// SIMATIC STEP 7 (V5.x) project PLC_DVG
// CPU: CPU 317-2 PN/DP
// station: Hardware
// station: SIMATIC 300 Station
// station: P_ADR_BUS
// station: _S7H_BUSSYSTEM_CT
// program: S7 Program(2)

SYMBOL_TABLE
"netsend"	DB 1000	DB 1000
"DI_DO_STATE"	FB 1	FB 1
"TCON"	FB 65	FB 65	// Connect
"TCP_MB_CLIENT"	FB 70	FB 70
"TCP_MB_SERVER"	FB 71	FB 71
"DO_MANUAL"	FC 1	FC 1
"sp_nm11"	I 0.0	BOOL
"md_znm12"	I 0.1	BOOL
"md_nm11"	I 0.2	BOOL
"tz_znm12"	I 0.3	BOOL
"tz_nm11"	I 0.4	BOOL
"sp_nm13"	I 0.5	BOOL
"sp_znm12"	I 0.6	BOOL
"md_nm13"	I 0.7	BOOL
"tz_nm13"	I 1.0	BOOL
"alm_znm15"	I 1.1	BOOL
"sp_nm14"	I 1.2	BOOL
"md_znm15"	I 1.3	BOOL
"md_nm14"	I 1.4	BOOL
"tz_nm14"	I 1.6	BOOL
"md_nm16"	I 2.0	BOOL
"tz_nm17_1"	I 2.1	BOOL
"tz_nm16"	I 2.2	BOOL
"sp_nm17_1"	I 2.4	BOOL
"md_nm17_2"	I 2.5	BOOL
"md_nm17_1"	I 2.6	BOOL
"tz_nm17_2"	I 2.7	BOOL
"sp_nm18"	I 3.0	BOOL
"md_nm19"	I 3.1	BOOL
"md_nm18"	I 3.2	BOOL
"tz_nm19"	I 3.3	BOOL
"tz_nm18"	I 3.4	BOOL
"md_nm19_1"	I 3.7	BOOL
"tz_nm19_1"	I 4.0	BOOL
"sp_no21"	I 4.1	BOOL
"sp_nm20"	I 4.2	BOOL
"md_no21"	I 4.3	BOOL
"md_nm20"	I 4.4	BOOL
"tz_no21"	I 4.5	BOOL
"tz_nm20"	I 4.6	BOOL
"md_no22"	I 5.0	BOOL
"av_vn2"	I 5.1	BOOL
"tz_no22"	I 5.2	BOOL
"md_vn1"	I 5.3	BOOL
"md_vn2"	I 5.4	BOOL
"tz_vn1"	I 5.5	BOOL
"tz_vn2"	I 5.6	BOOL
"sp_vn1"	I 5.7	BOOL
"av_vn1"	I 6.0	BOOL
"md_nv23"	I 6.1	BOOL
"tz_nv23"	I 6.3	BOOL
"temp_vn1"	I 6.4	BOOL
"sp_nv23_1"	I 6.5	BOOL
"sp_nv23"	I 6.6	BOOL
"md_nv23_1"	I 6.7	BOOL
"tz_nv23_1"	I 7.0	BOOL
"sp_nv25"	I 7.1	BOOL
"sp_nm24"	I 7.2	BOOL
"md_nv25"	I 7.3	BOOL
"md_nm24"	I 7.4	BOOL
"tz_nv25"	I 7.5	BOOL
"tz_nm24"	I 7.6	BOOL
"sp_nv26"	I 7.7	BOOL
"md_nv26"	I 8.0	BOOL
"tz_nv27"	I 8.1	BOOL
"tz_nv26"	I 8.2	BOOL
"sp_nv28"	I 8.3	BOOL
"sp_nv27"	I 8.4	BOOL
"md_nv28"	I 8.5	BOOL
"md_nv27"	I 8.6	BOOL
"tz_nv28"	I 8.7	BOOL
"md_nm30"	I 9.1	BOOL
"md_nv29"	I 9.2	BOOL
"tz_nm30"	I 9.3	BOOL
"tz_nv29"	I 9.4	BOOL
"sp_nm31"	I 9.5	BOOL
"md_nm31"	I 9.7	BOOL
"tz_nm31"	I 10.0	BOOL
"md_nc33"	I 10.3	BOOL
"md_nc32"	I 10.4	BOOL
"tz_nc33"	I 10.5	BOOL
"tz_nc32"	I 10.6	BOOL
"sp_nc34"	I 10.7	BOOL
"md_nc34"	I 11.0	BOOL
"tz_nc35"	I 11.1	BOOL
"tz_nc34"	I 11.2	BOOL
"sp_nc35"	I 11.4	BOOL
"md_nc33_1"	I 11.5	BOOL
"md_nc35"	I 11.6	BOOL
"tz_nc33_1"	I 11.7	BOOL
"md_vn3"	I 12.0	BOOL
"tz_vn3"	I 12.2	BOOL
"temp_vn3"	I 12.3	BOOL
"sp_vn3"	I 12.4	BOOL
"av_vn3"	I 12.6	BOOL
"md_dm2"	I 12.7	BOOL
"tz_dm2"	I 13.0	BOOL
"sp_m5"	I 13.1	BOOL
"sp_m4"	I 13.2	BOOL
"md_m5"	I 13.3	BOOL
"md_m4"	I 13.4	BOOL
"tz_m5"	I 13.5	BOOL
"tz_m4"	I 13.6	BOOL
"sp_m6"	I 13.7	BOOL
"md_m6"	I 14.0	BOOL
"tz_m6"	I 14.2	BOOL
"sp_m7"	I 14.4	BOOL
"md_m8"	I 14.5	BOOL
"md_m7"	I 14.6	BOOL
"tz_m8"	I 14.7	BOOL
"sp_c8"	I 15.0	BOOL
"md_c9"	I 15.1	BOOL
"md_c8"	I 15.2	BOOL
"tz_c9"	I 15.3	BOOL
"tz_c8"	I 15.4	BOOL
"sp_c9"	I 15.6	BOOL
"md_ds3"	I 15.7	BOOL
"sp_ds3"	I 16.0	BOOL
"sp_em3"	I 16.1	BOOL
"md_em3"	I 16.3	BOOL
"md_ft1"	I 16.4	BOOL
"tz_em3"	I 16.5	BOOL
"tz_ft1"	I 16.6	BOOL
"md_d2"	I 17.0	BOOL
"tz_vv6"	I 17.1	BOOL
"tz_d2"	I 17.2	BOOL
"sp_zm2"	I 17.3	BOOL
"sp_vv6"	I 17.4	BOOL
"md_zm2"	I 17.5	BOOL
"md_vv6"	I 17.6	BOOL
"tz_zm2"	I 17.7	BOOL
"sp_vd1"	I 18.0	BOOL
"tz_vn5"	I 18.1	BOOL
"md_vd1"	I 18.2	BOOL
"sp_vn5"	I 18.3	BOOL
"tz_vd1"	I 18.4	BOOL
"av_vn5"	I 18.5	BOOL
"md_vn5"	I 18.6	BOOL
"temp_vn5"	I 19.0	BOOL
"sp_vd3"	I 19.1	BOOL
"sp_vd2"	I 19.2	BOOL
"md_vd3"	I 19.3	BOOL
"md_vd2"	I 19.4	BOOL
"tz_vd3"	I 19.5	BOOL
"tz_vd2"	I 19.6	BOOL
"sp_vd4"	I 19.7	BOOL
"md_vd4"	I 20.0	BOOL
"tz_vd5"	I 20.1	BOOL
"tz_vd4"	I 20.2	BOOL
"sp_vd6"	I 20.3	BOOL
"md_vd6"	I 20.5	BOOL
"md_vd5"	I 20.6	BOOL
"tz_vd6"	I 20.7	BOOL
"md_vn4"	I 24.5	BOOL
"tz_vn4"	I 24.7	BOOL
"sp_vn4"	I 25.0	BOOL
"av_vn4"	I 25.2	BOOL
"ZNM15_manual"	M 2000.1	BOOL
"ZNM12_manual"	M 2000.2	BOOL
"ZNM12_pusk_nya"	M 4116.0	BOOL
"ZNM12_stop_nya"	M 4116.1	BOOL
"ZNM15_pusk_nya"	M 4116.2	BOOL
"ZNM15_stop_nya"	M 4116.3	BOOL
"tstArray[0]"	MB 5000	BYTE
"tstArray[1]"	MB 5001	BYTE
"tstArray[2]"	MB 5002	BYTE
"tstArray[3]"	MB 5003	BYTE
"QNM11"	Q 0.0	BOOL
"QZNM15"	Q 0.1	BOOL
"QZNM12"	Q 0.2	BOOL
"QNM16"	Q 0.3	BOOL
"QNM13"	Q 0.4	BOOL
"QNM17_1"	Q 0.5	BOOL
"QNM14"	Q 0.6	BOOL
"QNM17_2"	Q 0.7	BOOL
"QNM18"	Q 1.0	BOOL
"QNO21"	Q 1.1	BOOL
"QNM19"	Q 1.2	BOOL
"QNO22"	Q 1.3	BOOL
"QNM19_1"	Q 1.4	BOOL
"QVN2"	Q 1.5	BOOL
"QNM20"	Q 1.6	BOOL
"QVN1"	Q 1.7	BOOL
"QNV23"	Q 2.0	BOOL
"QNV26"	Q 2.1	BOOL
"QNV23_1"	Q 2.2	BOOL
"QNV27"	Q 2.3	BOOL
"QNM24"	Q 2.4	BOOL
"QNV28"	Q 2.5	BOOL
"QNV25"	Q 2.6	BOOL
"QNV29"	Q 2.7	BOOL
"QNM30"	Q 3.0	BOOL
"QNC34"	Q 3.1	BOOL
"QNM31"	Q 3.2	BOOL
"QNC35"	Q 3.3	BOOL
"QNC32"	Q 3.4	BOOL
"QNC33_1"	Q 3.5	BOOL
"QNC33"	Q 3.6	BOOL
"QVN3"	Q 3.7	BOOL
"QDM2"	Q 4.0	BOOL
"QM7"	Q 4.1	BOOL
"QM4"	Q 4.2	BOOL
"QM8"	Q 4.3	BOOL
"QM5"	Q 4.4	BOOL
"QC8"	Q 4.5	BOOL
"QM6"	Q 4.6	BOOL
"QC9"	Q 4.7	BOOL
"QDS3"	Q 5.0	BOOL
"QVV6"	Q 5.1	BOOL
"QFT1"	Q 5.2	BOOL
"QZM2"	Q 5.3	BOOL
"QEM3"	Q 5.4	BOOL
"QVD1"	Q 5.5	BOOL
"QD2"	Q 5.6	BOOL
"QVN5"	Q 5.7	BOOL
"QVD2"	Q 6.0	BOOL
"QVD6"	Q 6.1	BOOL
"QVD3"	Q 6.2	BOOL
"QVD4"	Q 6.4	BOOL
"QVD5"	Q 6.6	BOOL
"QVN4"	Q 7.7	BOOL
"TON"	SFB 4	SFB 4	// Generate an On Delay
"GET"	SFB 14	SFB 14	// Read Data From a Remote CPU
"PUT"	SFB 15	SFB 15	// Write Data to a Remote CPU
"VAT_DVG_ALL"	VAT 1	
"VAT_2"	VAT 2	
"VAT_3"	VAT 3	
END_SYMBOL_TABLE

FUNCTION_BLOCK "DI_DO_STATE"	// FB 1
TITLE = DI_DO_STATE
//Состояние дискретных входов PLC_DVG для SCADA
VERSION : 0.1
BEGIN
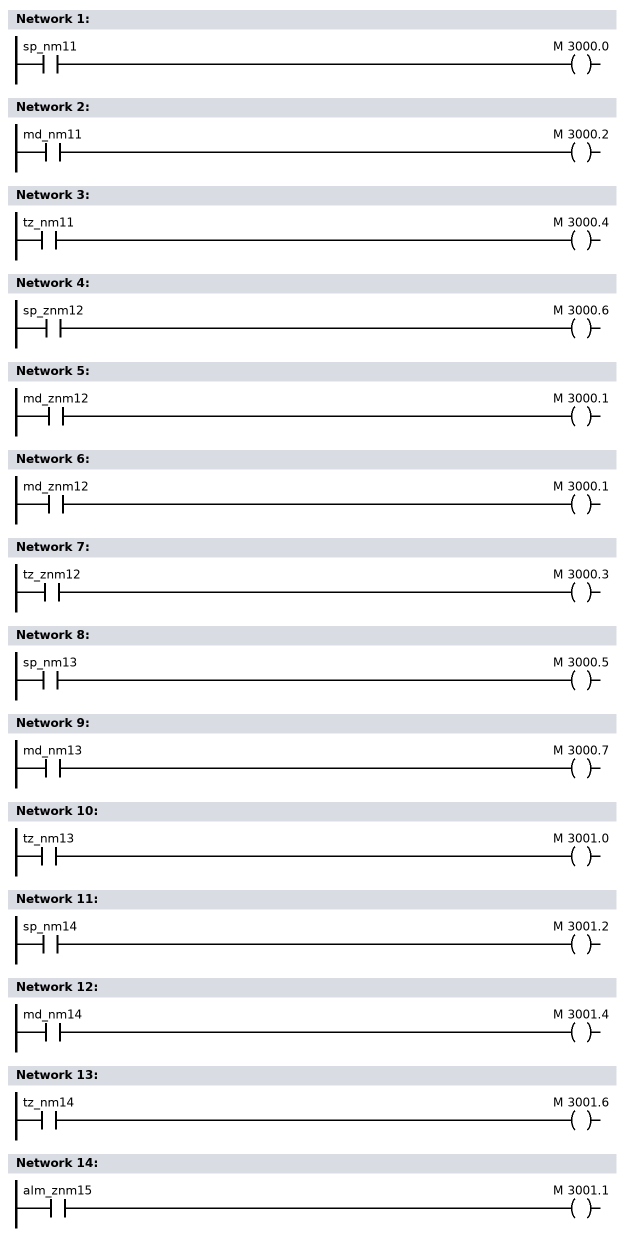
NETWORK
TITLE =
      A     "sp_nm11";
      =     M 3000.0;
NETWORK
TITLE =
      A     "md_nm11";
      =     M 3000.2;
NETWORK
TITLE =
      A     "tz_nm11";
      =     M 3000.4;
NETWORK
TITLE =
      A     "sp_znm12";
      =     M 3000.6;
NETWORK
TITLE =
      A     "md_znm12";
      =     M 3000.1;
NETWORK
TITLE =
      A     "md_znm12";
      =     M 3000.1;
NETWORK
TITLE =
      A     "tz_znm12";
      =     M 3000.3;
NETWORK
TITLE =
      A     "sp_nm13";
      =     M 3000.5;
NETWORK
TITLE =
      A     "md_nm13";
      =     M 3000.7;
NETWORK
TITLE =
      A     "tz_nm13";
      =     M 3001.0;
NETWORK
TITLE =
      A     "sp_nm14";
      =     M 3001.2;
NETWORK
TITLE =
      A     "md_nm14";
      =     M 3001.4;
NETWORK
TITLE =
      A     "tz_nm14";
      =     M 3001.6;
NETWORK
TITLE =
      A     "alm_znm15";
      =     M 3001.1;
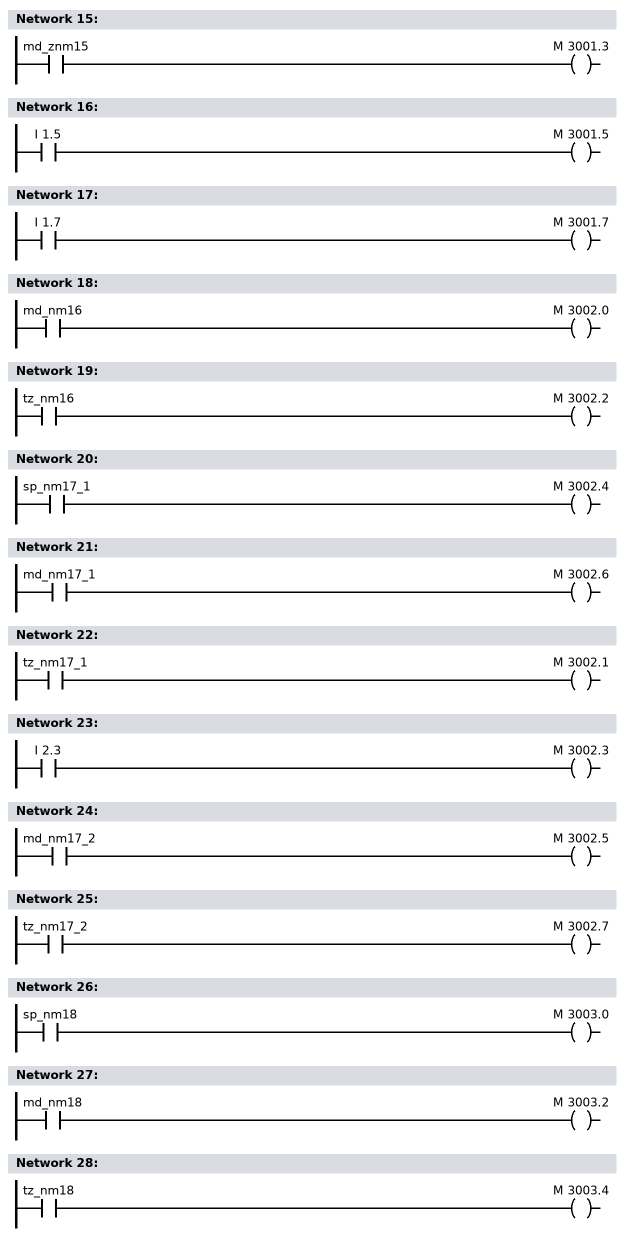
NETWORK
TITLE =
      A     "md_znm15";
      =     M 3001.3;
NETWORK
TITLE =
      A     I 1.5;
      =     M 3001.5;
NETWORK
TITLE =
      A     I 1.7;
      =     M 3001.7;
NETWORK
TITLE =
      A     "md_nm16";
      =     M 3002.0;
NETWORK
TITLE =
      A     "tz_nm16";
      =     M 3002.2;
NETWORK
TITLE =
      A     "sp_nm17_1";
      =     M 3002.4;
NETWORK
TITLE =
      A     "md_nm17_1";
      =     M 3002.6;
NETWORK
TITLE =
      A     "tz_nm17_1";
      =     M 3002.1;
NETWORK
TITLE =
      A     I 2.3;
      =     M 3002.3;
NETWORK
TITLE =
      A     "md_nm17_2";
      =     M 3002.5;
NETWORK
TITLE =
      A     "tz_nm17_2";
      =     M 3002.7;
NETWORK
TITLE =
      A     "sp_nm18";
      =     M 3003.0;
NETWORK
TITLE =
      A     "md_nm18";
      =     M 3003.2;
NETWORK
TITLE =
      A     "tz_nm18";
      =     M 3003.4;
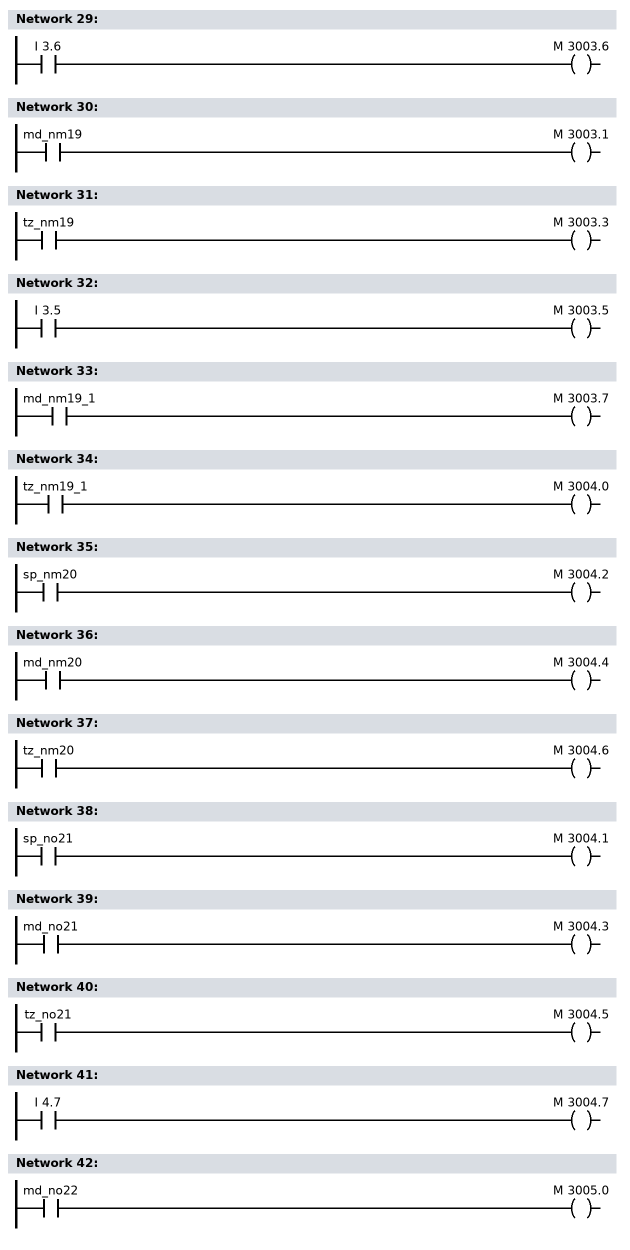
NETWORK
TITLE =
      A     I 3.6;
      =     M 3003.6;
NETWORK
TITLE =
      A     "md_nm19";
      =     M 3003.1;
NETWORK
TITLE =
      A     "tz_nm19";
      =     M 3003.3;
NETWORK
TITLE =
      A     I 3.5;
      =     M 3003.5;
NETWORK
TITLE =
      A     "md_nm19_1";
      =     M 3003.7;
NETWORK
TITLE =
      A     "tz_nm19_1";
      =     M 3004.0;
NETWORK
TITLE =
      A     "sp_nm20";
      =     M 3004.2;
NETWORK
TITLE =
      A     "md_nm20";
      =     M 3004.4;
NETWORK
TITLE =
      A     "tz_nm20";
      =     M 3004.6;
NETWORK
TITLE =
      A     "sp_no21";
      =     M 3004.1;
NETWORK
TITLE =
      A     "md_no21";
      =     M 3004.3;
NETWORK
TITLE =
      A     "tz_no21";
      =     M 3004.5;
NETWORK
TITLE =
      A     I 4.7;
      =     M 3004.7;
NETWORK
TITLE =
      A     "md_no22";
      =     M 3005.0;
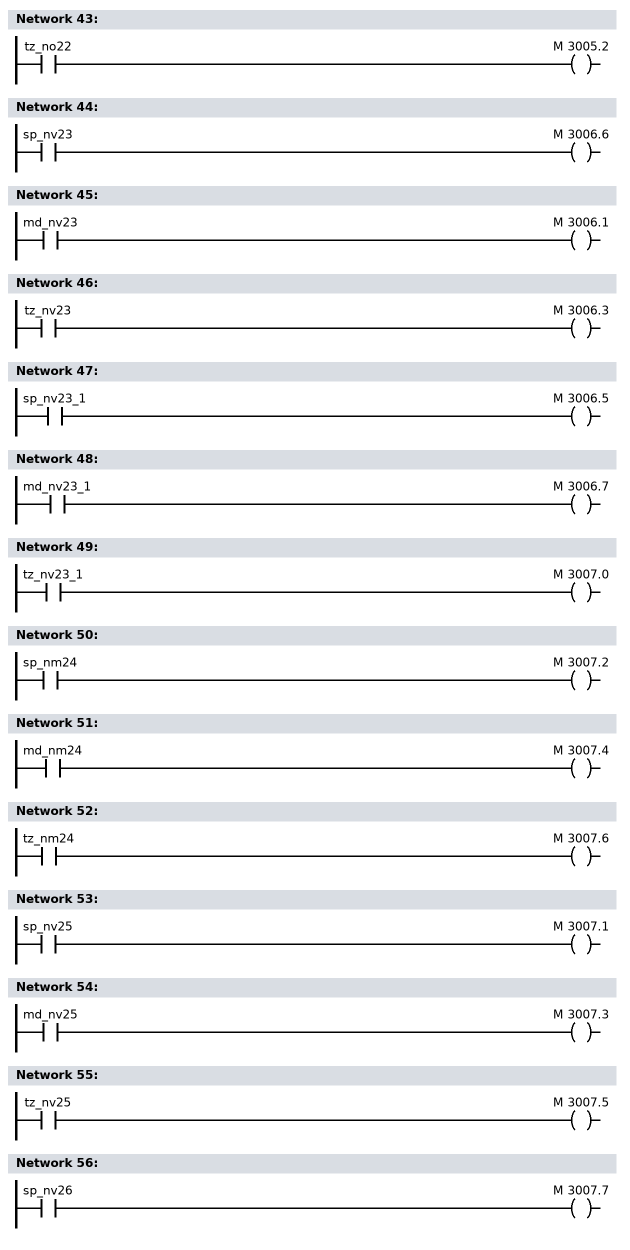
NETWORK
TITLE =
      A     "tz_no22";
      =     M 3005.2;
NETWORK
TITLE =
      A     "sp_nv23";
      =     M 3006.6;
NETWORK
TITLE =
      A     "md_nv23";
      =     M 3006.1;
NETWORK
TITLE =
      A     "tz_nv23";
      =     M 3006.3;
NETWORK
TITLE =
      A     "sp_nv23_1";
      =     M 3006.5;
NETWORK
TITLE =
      A     "md_nv23_1";
      =     M 3006.7;
NETWORK
TITLE =
      A     "tz_nv23_1";
      =     M 3007.0;
NETWORK
TITLE =
      A     "sp_nm24";
      =     M 3007.2;
NETWORK
TITLE =
      A     "md_nm24";
      =     M 3007.4;
NETWORK
TITLE =
      A     "tz_nm24";
      =     M 3007.6;
NETWORK
TITLE =
      A     "sp_nv25";
      =     M 3007.1;
NETWORK
TITLE =
      A     "md_nv25";
      =     M 3007.3;
NETWORK
TITLE =
      A     "tz_nv25";
      =     M 3007.5;
NETWORK
TITLE =
      A     "sp_nv26";
      =     M 3007.7;
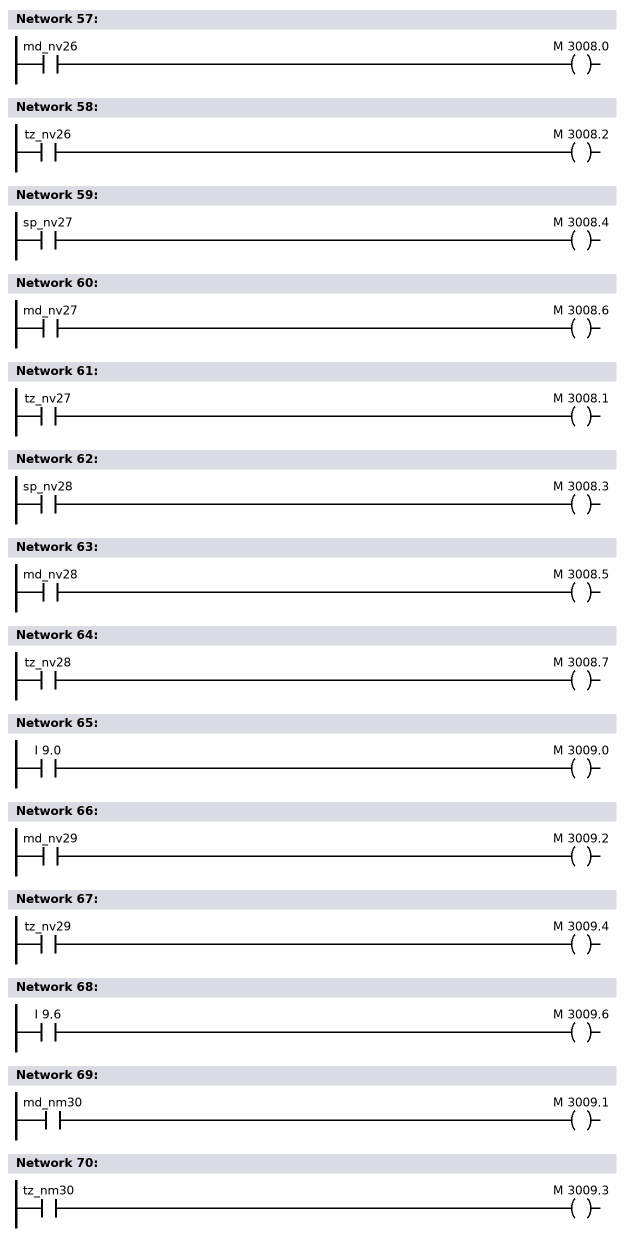
NETWORK
TITLE =
      A     "md_nv26";
      =     M 3008.0;
NETWORK
TITLE =
      A     "tz_nv26";
      =     M 3008.2;
NETWORK
TITLE =
      A     "sp_nv27";
      =     M 3008.4;
NETWORK
TITLE =
      A     "md_nv27";
      =     M 3008.6;
NETWORK
TITLE =
      A     "tz_nv27";
      =     M 3008.1;
NETWORK
TITLE =
      A     "sp_nv28";
      =     M 3008.3;
NETWORK
TITLE =
      A     "md_nv28";
      =     M 3008.5;
NETWORK
TITLE =
      A     "tz_nv28";
      =     M 3008.7;
NETWORK
TITLE =
      A     I 9.0;
      =     M 3009.0;
NETWORK
TITLE =
      A     "md_nv29";
      =     M 3009.2;
NETWORK
TITLE =
      A     "tz_nv29";
      =     M 3009.4;
NETWORK
TITLE =
      A     I 9.6;
      =     M 3009.6;
NETWORK
TITLE =
      A     "md_nm30";
      =     M 3009.1;
NETWORK
TITLE =
      A     "tz_nm30";
      =     M 3009.3;
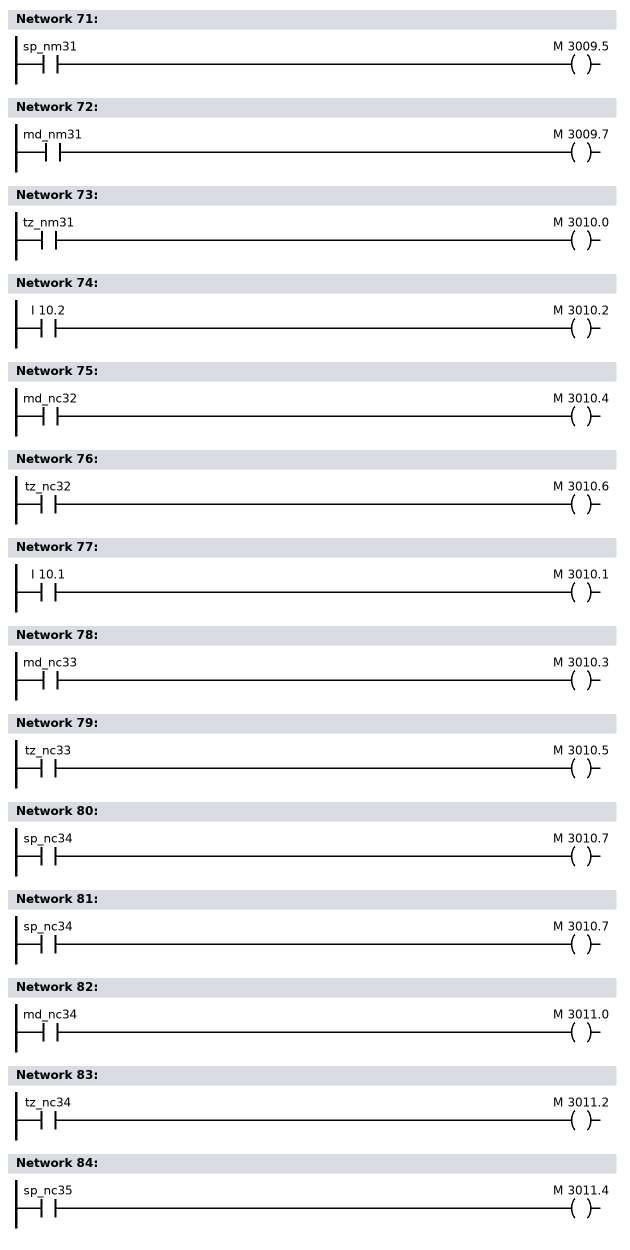
NETWORK
TITLE =
      A     "sp_nm31";
      =     M 3009.5;
NETWORK
TITLE =
      A     "md_nm31";
      =     M 3009.7;
NETWORK
TITLE =
      A     "tz_nm31";
      =     M 3010.0;
NETWORK
TITLE =
      A     I 10.2;
      =     M 3010.2;
NETWORK
TITLE =
      A     "md_nc32";
      =     M 3010.4;
NETWORK
TITLE =
      A     "tz_nc32";
      =     M 3010.6;
NETWORK
TITLE =
      A     I 10.1;
      =     M 3010.1;
NETWORK
TITLE =
      A     "md_nc33";
      =     M 3010.3;
NETWORK
TITLE =
      A     "tz_nc33";
      =     M 3010.5;
NETWORK
TITLE =
      A     "sp_nc34";
      =     M 3010.7;
NETWORK
TITLE =
      A     "sp_nc34";
      =     M 3010.7;
NETWORK
TITLE =
      A     "md_nc34";
      =     M 3011.0;
NETWORK
TITLE =
      A     "tz_nc34";
      =     M 3011.2;
NETWORK
TITLE =
      A     "sp_nc35";
      =     M 3011.4;
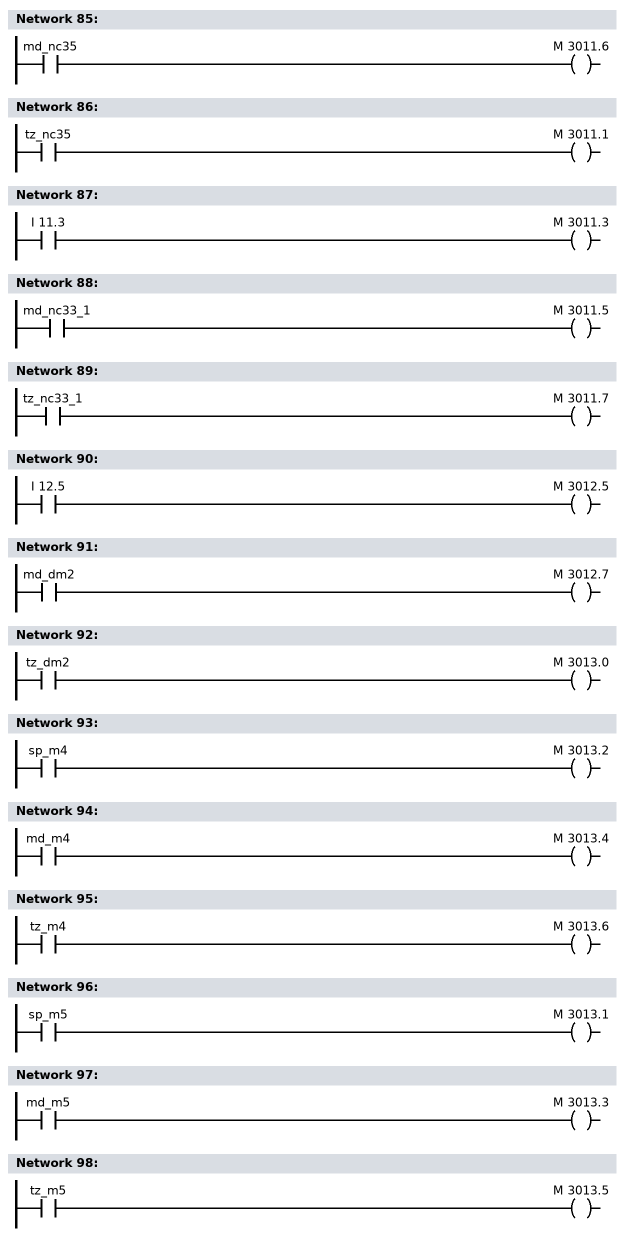
NETWORK
TITLE =
      A     "md_nc35";
      =     M 3011.6;
NETWORK
TITLE =
      A     "tz_nc35";
      =     M 3011.1;
NETWORK
TITLE =
      A     I 11.3;
      =     M 3011.3;
NETWORK
TITLE =
      A     "md_nc33_1";
      =     M 3011.5;
NETWORK
TITLE =
      A     "tz_nc33_1";
      =     M 3011.7;
NETWORK
TITLE =
      A     I 12.5;
      =     M 3012.5;
NETWORK
TITLE =
      A     "md_dm2";
      =     M 3012.7;
NETWORK
TITLE =
      A     "tz_dm2";
      =     M 3013.0;
NETWORK
TITLE =
      A     "sp_m4";
      =     M 3013.2;
NETWORK
TITLE =
      A     "md_m4";
      =     M 3013.4;
NETWORK
TITLE =
      A     "tz_m4";
      =     M 3013.6;
NETWORK
TITLE =
      A     "sp_m5";
      =     M 3013.1;
NETWORK
TITLE =
      A     "md_m5";
      =     M 3013.3;
NETWORK
TITLE =
      A     "tz_m5";
      =     M 3013.5;
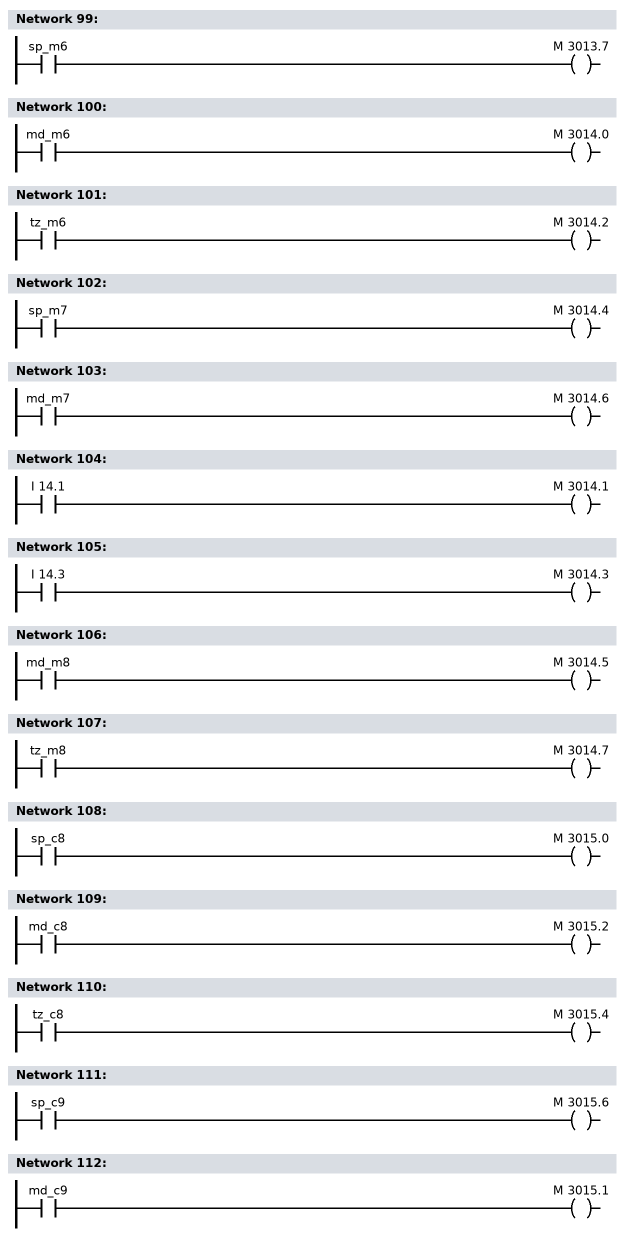
NETWORK
TITLE =
      A     "sp_m6";
      =     M 3013.7;
NETWORK
TITLE =
      A     "md_m6";
      =     M 3014.0;
NETWORK
TITLE =
      A     "tz_m6";
      =     M 3014.2;
NETWORK
TITLE =
      A     "sp_m7";
      =     M 3014.4;
NETWORK
TITLE =
      A     "md_m7";
      =     M 3014.6;
NETWORK
TITLE =
      A     I 14.1;
      =     M 3014.1;
NETWORK
TITLE =
      A     I 14.3;
      =     M 3014.3;
NETWORK
TITLE =
      A     "md_m8";
      =     M 3014.5;
NETWORK
TITLE =
      A     "tz_m8";
      =     M 3014.7;
NETWORK
TITLE =
      A     "sp_c8";
      =     M 3015.0;
NETWORK
TITLE =
      A     "md_c8";
      =     M 3015.2;
NETWORK
TITLE =
      A     "tz_c8";
      =     M 3015.4;
NETWORK
TITLE =
      A     "sp_c9";
      =     M 3015.6;
NETWORK
TITLE =
      A     "md_c9";
      =     M 3015.1;
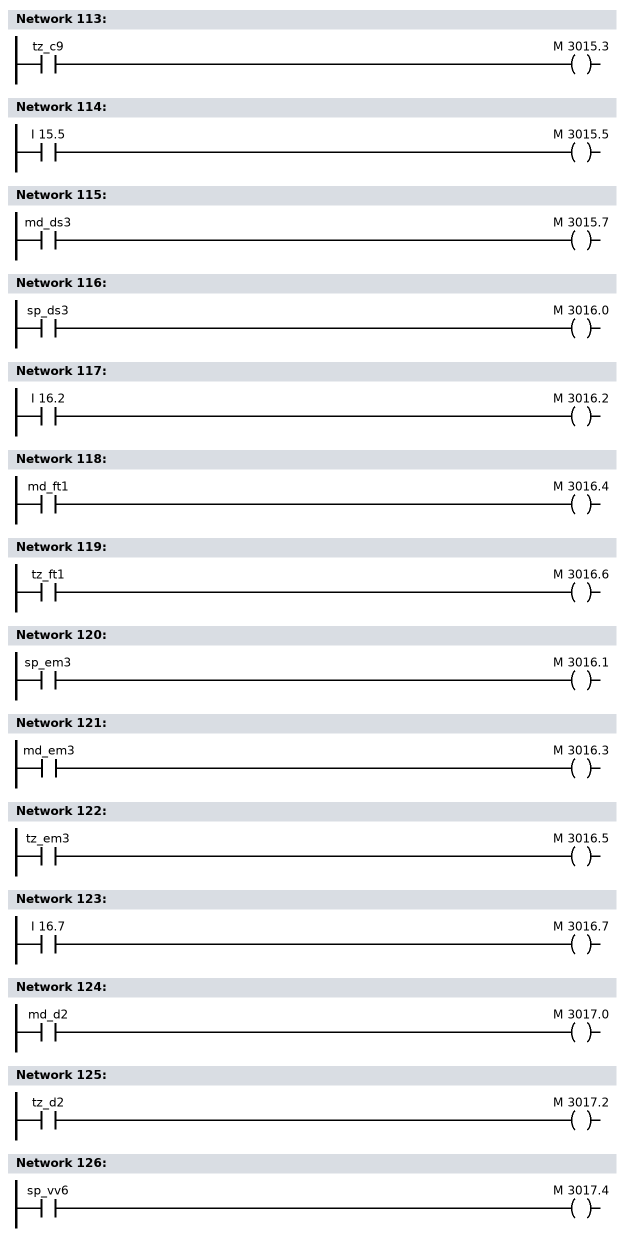
NETWORK
TITLE =
      A     "tz_c9";
      =     M 3015.3;
NETWORK
TITLE =
      A     I 15.5;
      =     M 3015.5;
NETWORK
TITLE =
      A     "md_ds3";
      =     M 3015.7;
NETWORK
TITLE =
      A     "sp_ds3";
      =     M 3016.0;
NETWORK
TITLE =
      A     I 16.2;
      =     M 3016.2;
NETWORK
TITLE =
      A     "md_ft1";
      =     M 3016.4;
NETWORK
TITLE =
      A     "tz_ft1";
      =     M 3016.6;
NETWORK
TITLE =
      A     "sp_em3";
      =     M 3016.1;
NETWORK
TITLE =
      A     "md_em3";
      =     M 3016.3;
NETWORK
TITLE =
      A     "tz_em3";
      =     M 3016.5;
NETWORK
TITLE =
      A     I 16.7;
      =     M 3016.7;
NETWORK
TITLE =
      A     "md_d2";
      =     M 3017.0;
NETWORK
TITLE =
      A     "tz_d2";
      =     M 3017.2;
NETWORK
TITLE =
      A     "sp_vv6";
      =     M 3017.4;
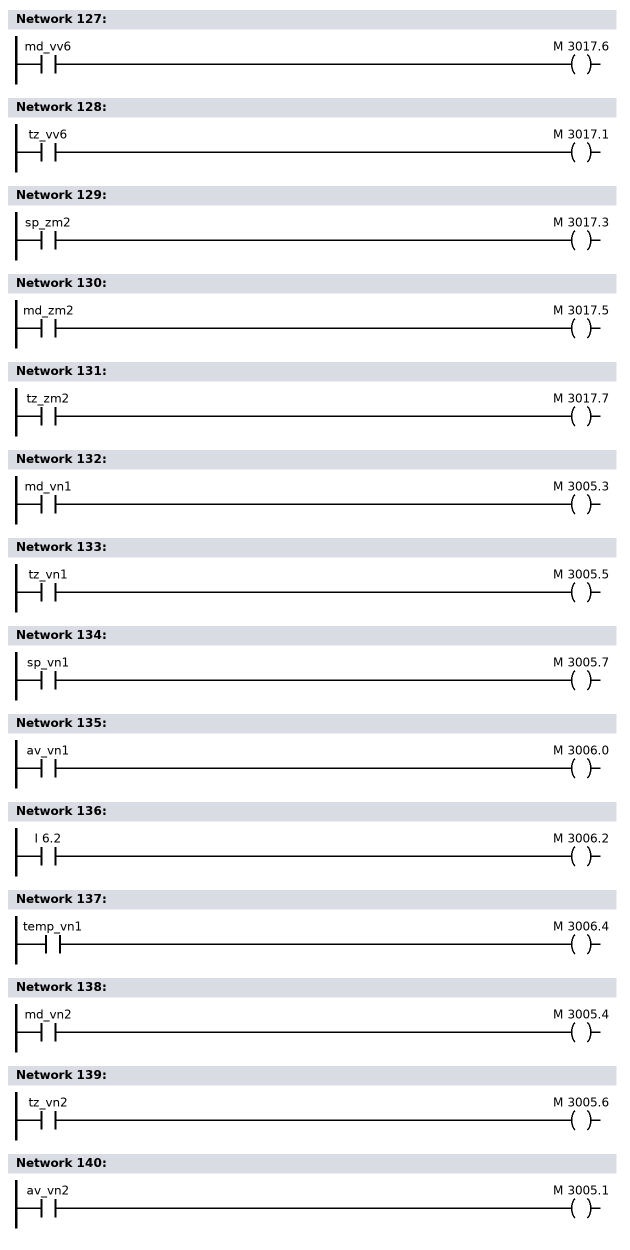
NETWORK
TITLE =
      A     "md_vv6";
      =     M 3017.6;
NETWORK
TITLE =
      A     "tz_vv6";
      =     M 3017.1;
NETWORK
TITLE =
      A     "sp_zm2";
      =     M 3017.3;
NETWORK
TITLE =
      A     "md_zm2";
      =     M 3017.5;
NETWORK
TITLE =
      A     "tz_zm2";
      =     M 3017.7;
NETWORK
TITLE =
      A     "md_vn1";
      =     M 3005.3;
NETWORK
TITLE =
      A     "tz_vn1";
      =     M 3005.5;
NETWORK
TITLE =
      A     "sp_vn1";
      =     M 3005.7;
NETWORK
TITLE =
      A     "av_vn1";
      =     M 3006.0;
NETWORK
TITLE =
      A     I 6.2;
      =     M 3006.2;
NETWORK
TITLE =
      A     "temp_vn1";
      =     M 3006.4;
NETWORK
TITLE =
      A     "md_vn2";
      =     M 3005.4;
NETWORK
TITLE =
      A     "tz_vn2";
      =     M 3005.6;
NETWORK
TITLE =
      A     "av_vn2";
      =     M 3005.1;
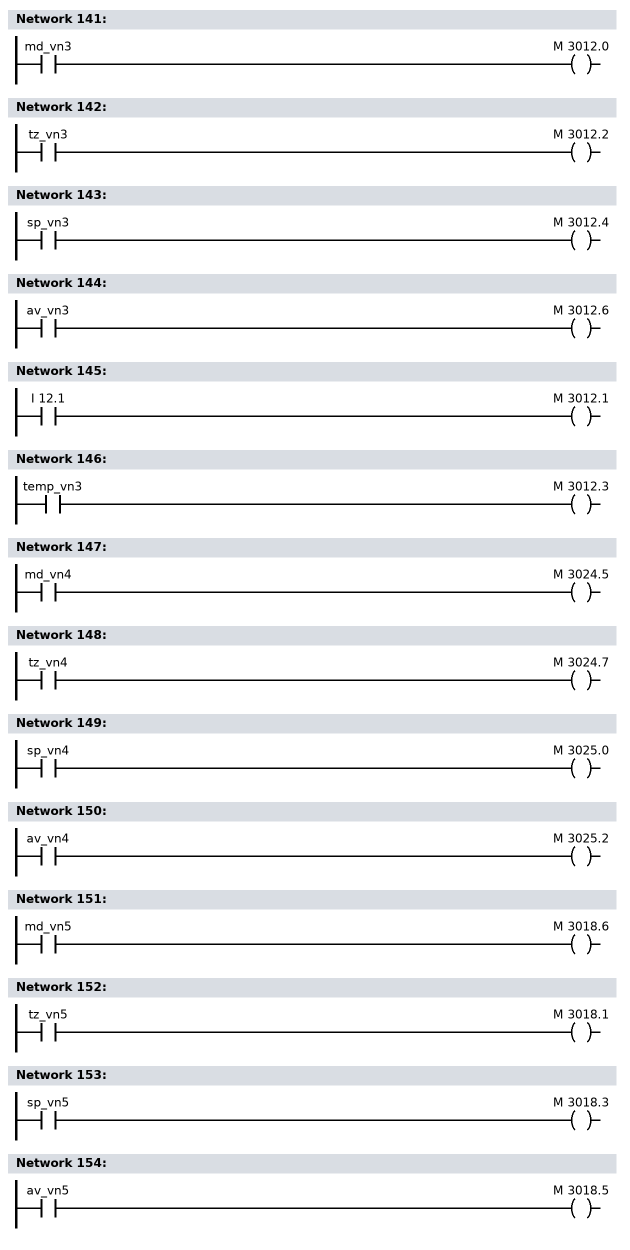
NETWORK
TITLE =
      A     "md_vn3";
      =     M 3012.0;
NETWORK
TITLE =
      A     "tz_vn3";
      =     M 3012.2;
NETWORK
TITLE =
      A     "sp_vn3";
      =     M 3012.4;
NETWORK
TITLE =
      A     "av_vn3";
      =     M 3012.6;
NETWORK
TITLE =
      A     I 12.1;
      =     M 3012.1;
NETWORK
TITLE =
      A     "temp_vn3";
      =     M 3012.3;
NETWORK
TITLE =
      A     "md_vn4";
      =     M 3024.5;
NETWORK
TITLE =
      A     "tz_vn4";
      =     M 3024.7;
NETWORK
TITLE =
      A     "sp_vn4";
      =     M 3025.0;
NETWORK
TITLE =
      A     "av_vn4";
      =     M 3025.2;
NETWORK
TITLE =
      A     "md_vn5";
      =     M 3018.6;
NETWORK
TITLE =
      A     "tz_vn5";
      =     M 3018.1;
NETWORK
TITLE =
      A     "sp_vn5";
      =     M 3018.3;
NETWORK
TITLE =
      A     "av_vn5";
      =     M 3018.5;
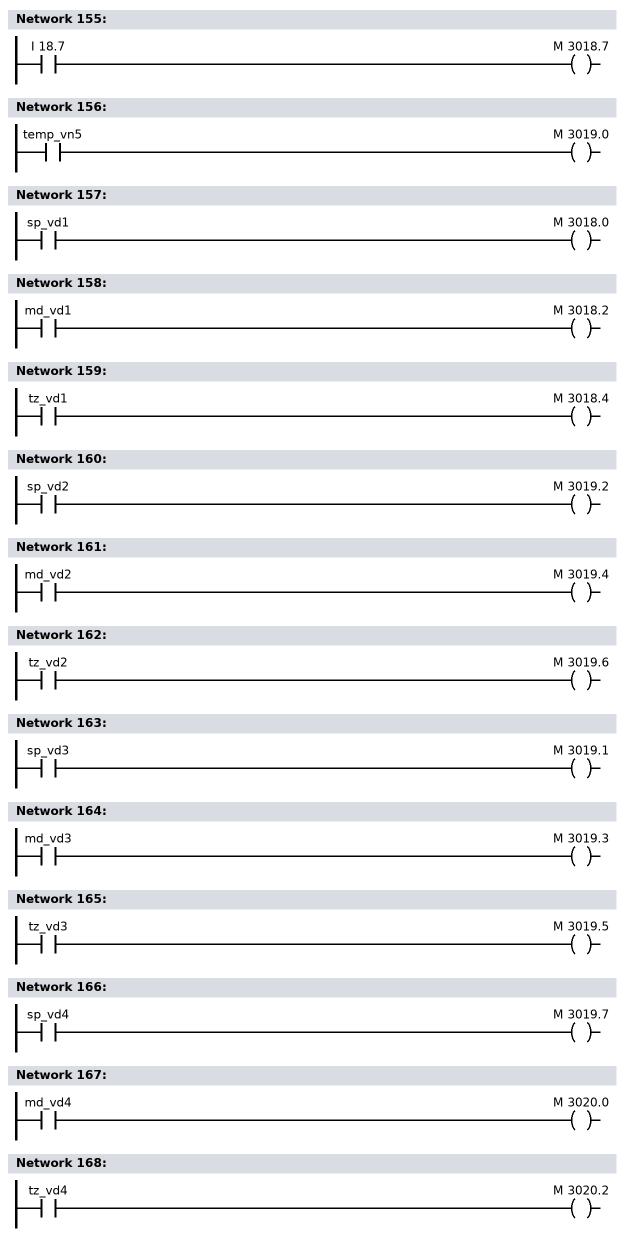
NETWORK
TITLE =
      A     I 18.7;
      =     M 3018.7;
NETWORK
TITLE =
      A     "temp_vn5";
      =     M 3019.0;
NETWORK
TITLE =
      A     "sp_vd1";
      =     M 3018.0;
NETWORK
TITLE =
      A     "md_vd1";
      =     M 3018.2;
NETWORK
TITLE =
      A     "tz_vd1";
      =     M 3018.4;
NETWORK
TITLE =
      A     "sp_vd2";
      =     M 3019.2;
NETWORK
TITLE =
      A     "md_vd2";
      =     M 3019.4;
NETWORK
TITLE =
      A     "tz_vd2";
      =     M 3019.6;
NETWORK
TITLE =
      A     "sp_vd3";
      =     M 3019.1;
NETWORK
TITLE =
      A     "md_vd3";
      =     M 3019.3;
NETWORK
TITLE =
      A     "tz_vd3";
      =     M 3019.5;
NETWORK
TITLE =
      A     "sp_vd4";
      =     M 3019.7;
NETWORK
TITLE =
      A     "md_vd4";
      =     M 3020.0;
NETWORK
TITLE =
      A     "tz_vd4";
      =     M 3020.2;
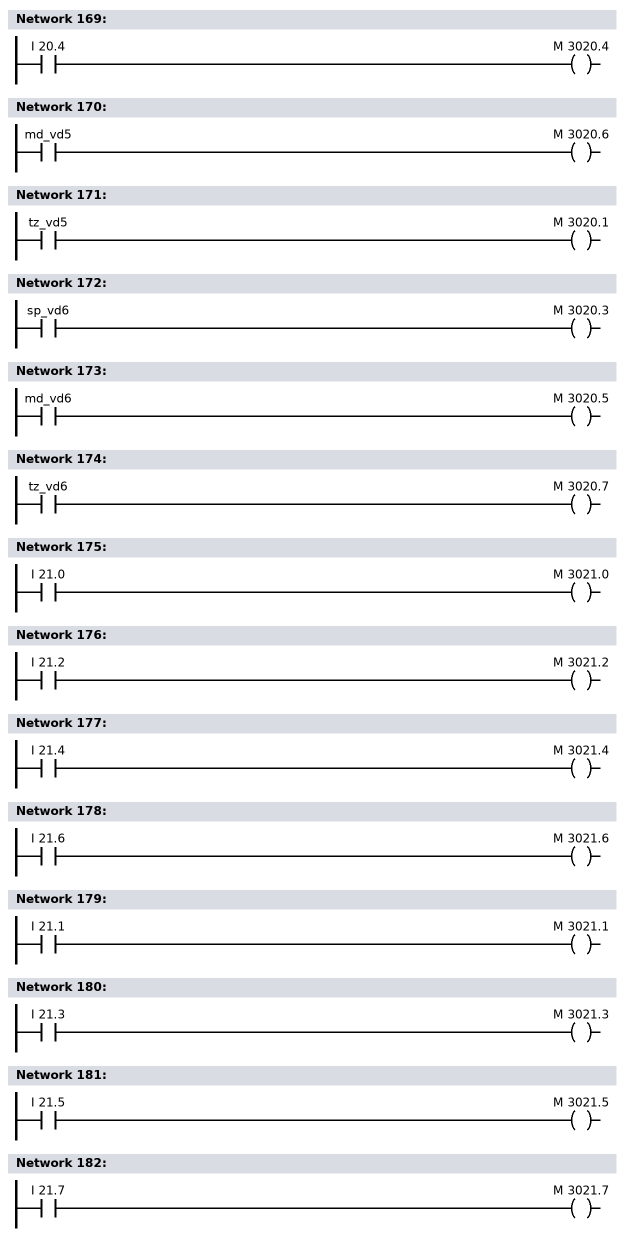
NETWORK
TITLE =
      A     I 20.4;
      =     M 3020.4;
NETWORK
TITLE =
      A     "md_vd5";
      =     M 3020.6;
NETWORK
TITLE =
      A     "tz_vd5";
      =     M 3020.1;
NETWORK
TITLE =
      A     "sp_vd6";
      =     M 3020.3;
NETWORK
TITLE =
      A     "md_vd6";
      =     M 3020.5;
NETWORK
TITLE =
      A     "tz_vd6";
      =     M 3020.7;
NETWORK
TITLE =
      A     I 21.0;
      =     M 3021.0;
NETWORK
TITLE =
      A     I 21.2;
      =     M 3021.2;
NETWORK
TITLE =
      A     I 21.4;
      =     M 3021.4;
NETWORK
TITLE =
      A     I 21.6;
      =     M 3021.6;
NETWORK
TITLE =
      A     I 21.1;
      =     M 3021.1;
NETWORK
TITLE =
      A     I 21.3;
      =     M 3021.3;
NETWORK
TITLE =
      A     I 21.5;
      =     M 3021.5;
NETWORK
TITLE =
      A     I 21.7;
      =     M 3021.7;
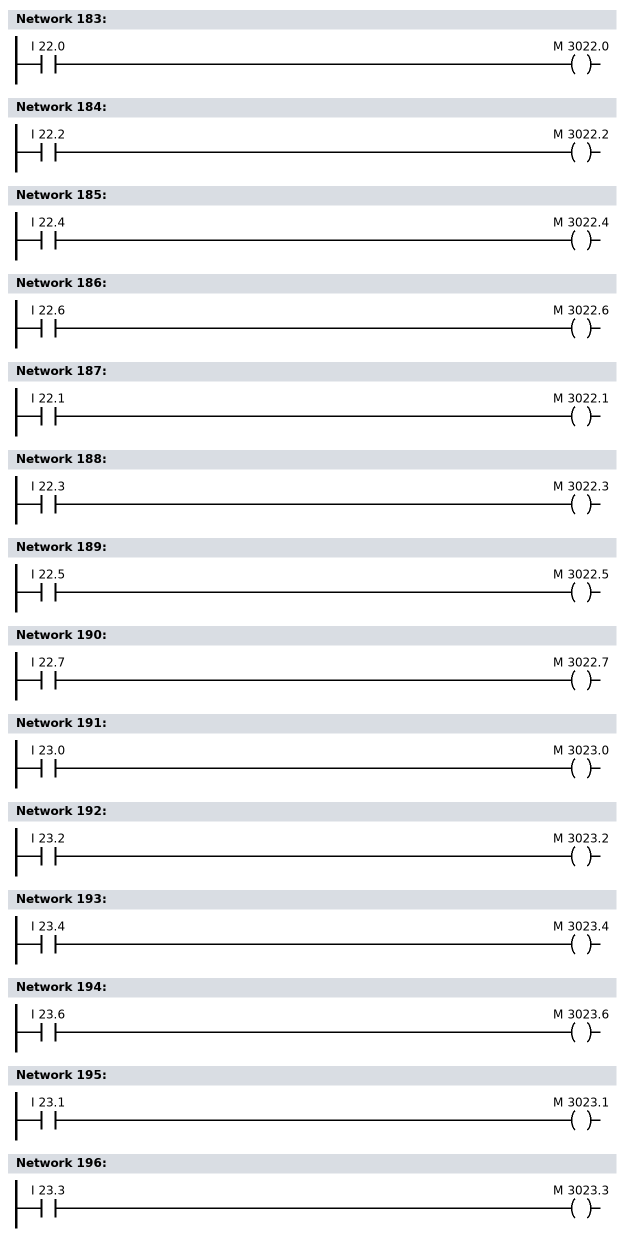
NETWORK
TITLE =
      A     I 22.0;
      =     M 3022.0;
NETWORK
TITLE =
      A     I 22.2;
      =     M 3022.2;
NETWORK
TITLE =
      A     I 22.4;
      =     M 3022.4;
NETWORK
TITLE =
      A     I 22.6;
      =     M 3022.6;
NETWORK
TITLE =
      A     I 22.1;
      =     M 3022.1;
NETWORK
TITLE =
      A     I 22.3;
      =     M 3022.3;
NETWORK
TITLE =
      A     I 22.5;
      =     M 3022.5;
NETWORK
TITLE =
      A     I 22.7;
      =     M 3022.7;
NETWORK
TITLE =
      A     I 23.0;
      =     M 3023.0;
NETWORK
TITLE =
      A     I 23.2;
      =     M 3023.2;
NETWORK
TITLE =
      A     I 23.4;
      =     M 3023.4;
NETWORK
TITLE =
      A     I 23.6;
      =     M 3023.6;
NETWORK
TITLE =
      A     I 23.1;
      =     M 3023.1;
NETWORK
TITLE =
      A     I 23.3;
      =     M 3023.3;
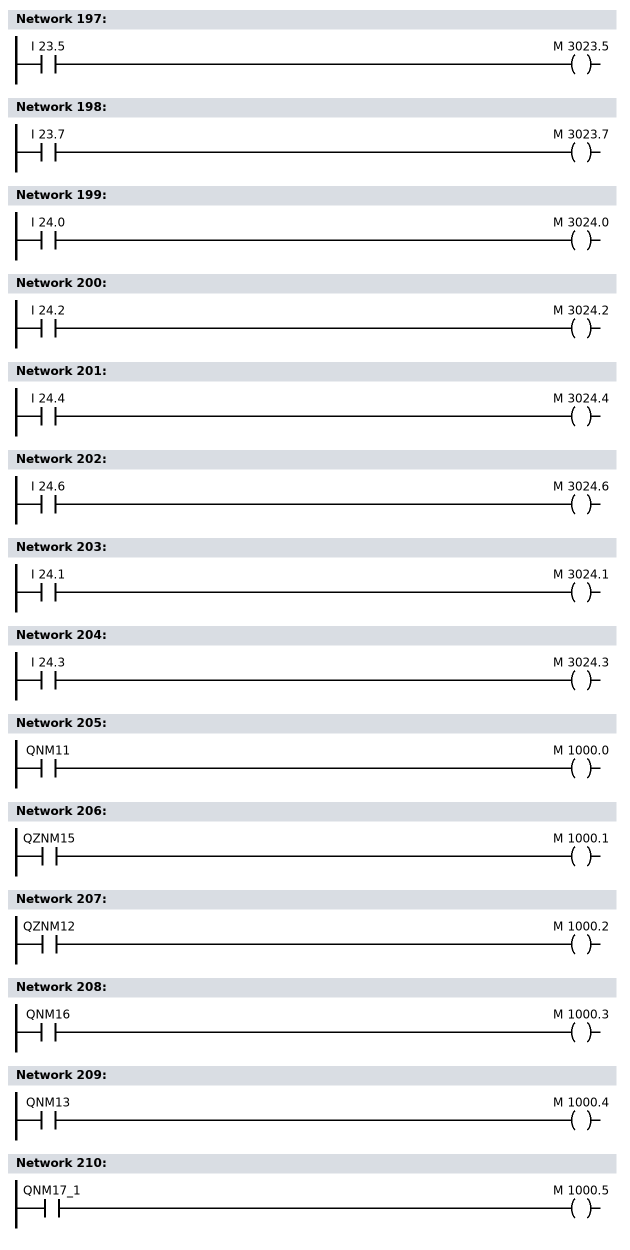
NETWORK
TITLE =
      A     I 23.5;
      =     M 3023.5;
NETWORK
TITLE =
      A     I 23.7;
      =     M 3023.7;
NETWORK
TITLE =
      A     I 24.0;
      =     M 3024.0;
NETWORK
TITLE =
      A     I 24.2;
      =     M 3024.2;
NETWORK
TITLE =
      A     I 24.4;
      =     M 3024.4;
NETWORK
TITLE =
      A     I 24.6;
      =     M 3024.6;
NETWORK
TITLE =
      A     I 24.1;
      =     M 3024.1;
NETWORK
TITLE =
      A     I 24.3;
      =     M 3024.3;
NETWORK
TITLE =
//Состояние дискретных выходов PLC_DVG для SCADA
      A     "QNM11";
      =     M 1000.0;
NETWORK
TITLE =
      A     "QZNM15";
      =     M 1000.1;
NETWORK
TITLE =
      A     "QZNM12";
      =     M 1000.2;
NETWORK
TITLE =
      A     "QNM16";
      =     M 1000.3;
NETWORK
TITLE =
      A     "QNM13";
      =     M 1000.4;
NETWORK
TITLE =
      A     "QNM17_1";
      =     M 1000.5;
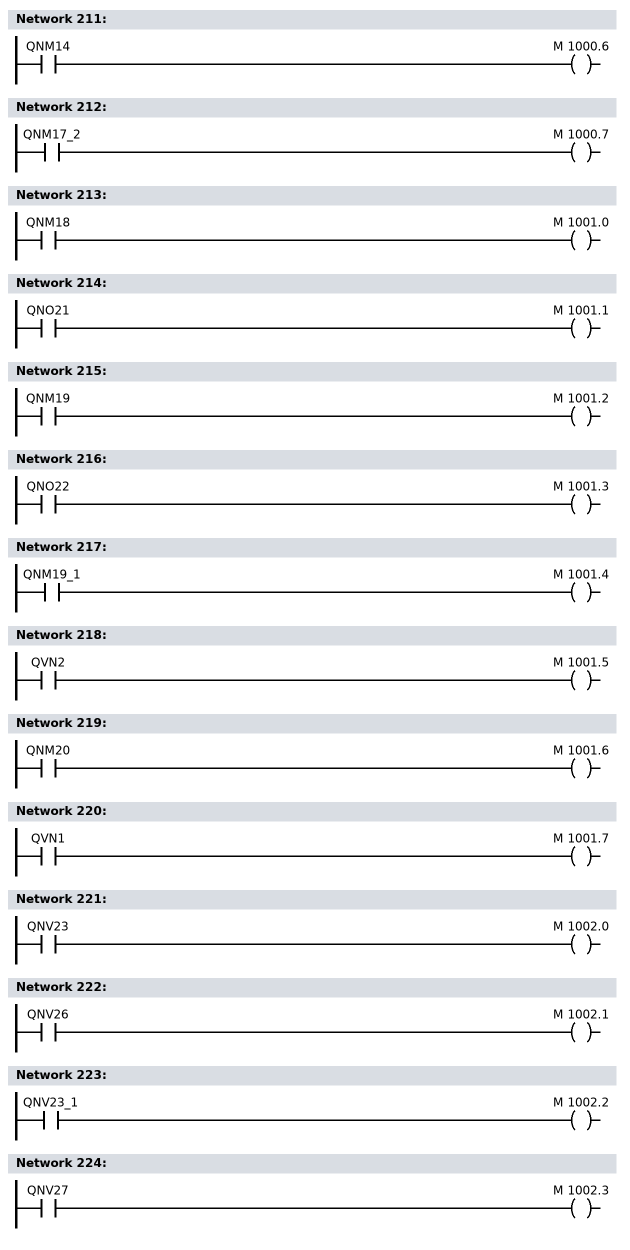
NETWORK
TITLE =
      A     "QNM14";
      =     M 1000.6;
NETWORK
TITLE =
      A     "QNM17_2";
      =     M 1000.7;
NETWORK
TITLE =
      A     "QNM18";
      =     M 1001.0;
NETWORK
TITLE =
      A     "QNO21";
      =     M 1001.1;
NETWORK
TITLE =
      A     "QNM19";
      =     M 1001.2;
NETWORK
TITLE =
      A     "QNO22";
      =     M 1001.3;
NETWORK
TITLE =
      A     "QNM19_1";
      =     M 1001.4;
NETWORK
TITLE =
      A     "QVN2";
      =     M 1001.5;
NETWORK
TITLE =
      A     "QNM20";
      =     M 1001.6;
NETWORK
TITLE =
      A     "QVN1";
      =     M 1001.7;
NETWORK
TITLE =
      A     "QNV23";
      =     M 1002.0;
NETWORK
TITLE =
      A     "QNV26";
      =     M 1002.1;
NETWORK
TITLE =
      A     "QNV23_1";
      =     M 1002.2;
NETWORK
TITLE =
      A     "QNV27";
      =     M 1002.3;
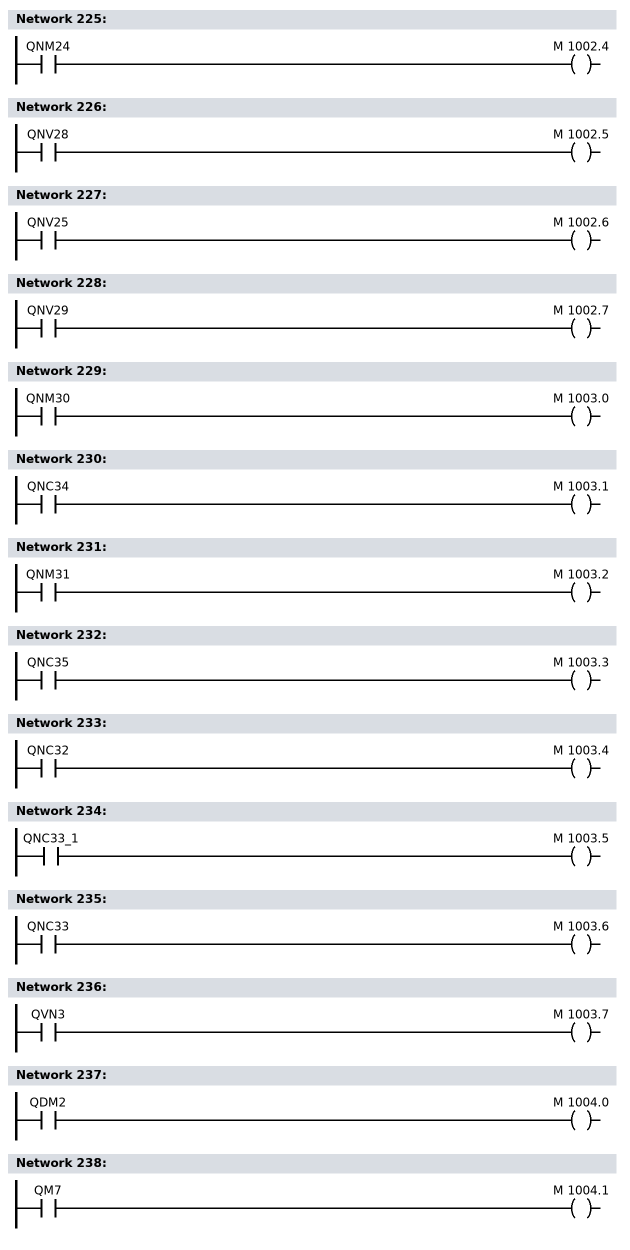
NETWORK
TITLE =
      A     "QNM24";
      =     M 1002.4;
NETWORK
TITLE =
      A     "QNV28";
      =     M 1002.5;
NETWORK
TITLE =
      A     "QNV25";
      =     M 1002.6;
NETWORK
TITLE =
      A     "QNV29";
      =     M 1002.7;
NETWORK
TITLE =
      A     "QNM30";
      =     M 1003.0;
NETWORK
TITLE =
      A     "QNC34";
      =     M 1003.1;
NETWORK
TITLE =
      A     "QNM31";
      =     M 1003.2;
NETWORK
TITLE =
      A     "QNC35";
      =     M 1003.3;
NETWORK
TITLE =
      A     "QNC32";
      =     M 1003.4;
NETWORK
TITLE =
      A     "QNC33_1";
      =     M 1003.5;
NETWORK
TITLE =
      A     "QNC33";
      =     M 1003.6;
NETWORK
TITLE =
      A     "QVN3";
      =     M 1003.7;
NETWORK
TITLE =
      A     "QDM2";
      =     M 1004.0;
NETWORK
TITLE =
      A     "QM7";
      =     M 1004.1;
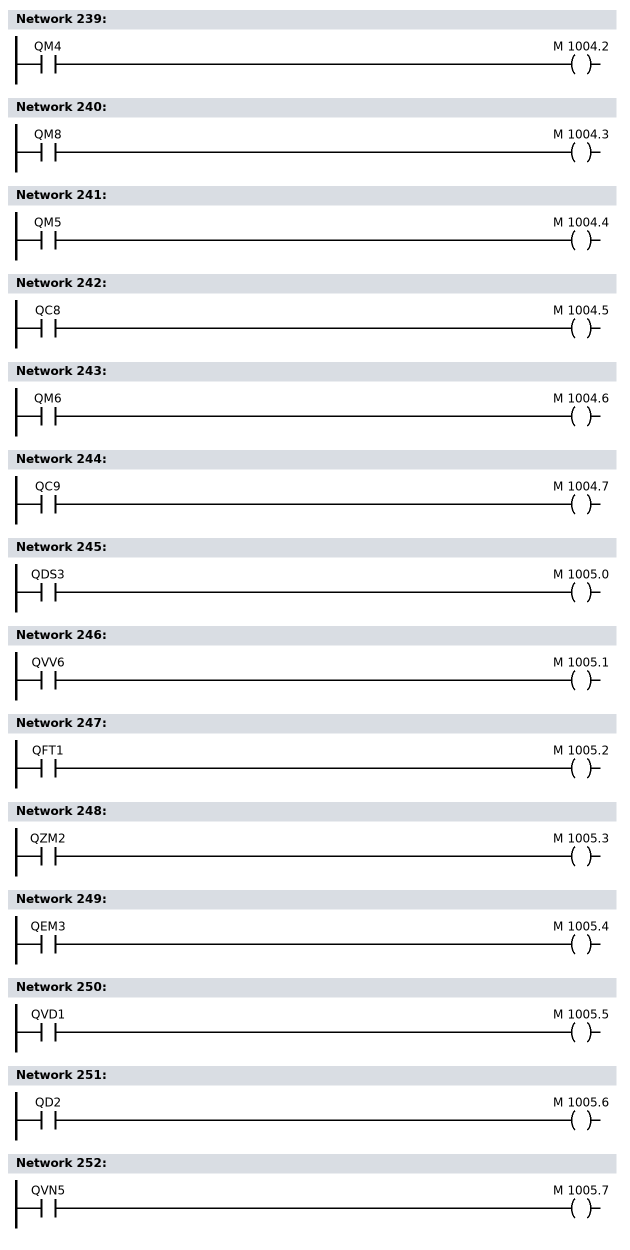
NETWORK
TITLE =
      A     "QM4";
      =     M 1004.2;
NETWORK
TITLE =
      A     "QM8";
      =     M 1004.3;
NETWORK
TITLE =
      A     "QM5";
      =     M 1004.4;
NETWORK
TITLE =
      A     "QC8";
      =     M 1004.5;
NETWORK
TITLE =
      A     "QM6";
      =     M 1004.6;
NETWORK
TITLE =
      A     "QC9";
      =     M 1004.7;
NETWORK
TITLE =
      A     "QDS3";
      =     M 1005.0;
NETWORK
TITLE =
      A     "QVV6";
      =     M 1005.1;
NETWORK
TITLE =
      A     "QFT1";
      =     M 1005.2;
NETWORK
TITLE =
      A     "QZM2";
      =     M 1005.3;
NETWORK
TITLE =
      A     "QEM3";
      =     M 1005.4;
NETWORK
TITLE =
      A     "QVD1";
      =     M 1005.5;
NETWORK
TITLE =
      A     "QD2";
      =     M 1005.6;
NETWORK
TITLE =
      A     "QVN5";
      =     M 1005.7;
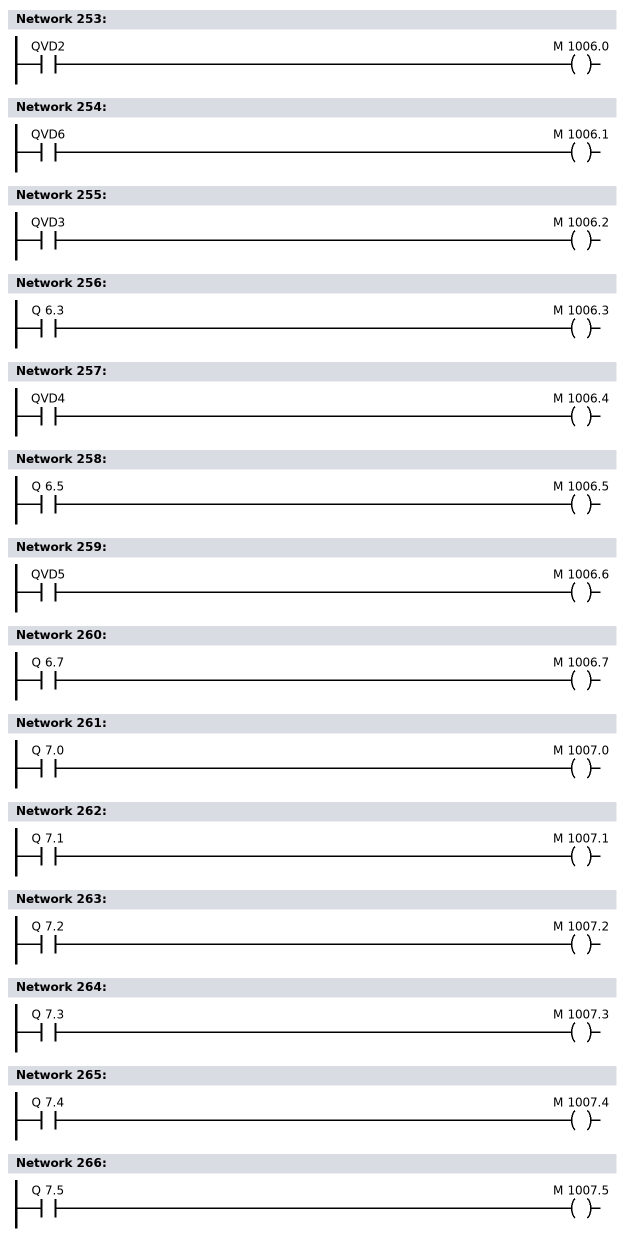
NETWORK
TITLE =
      A     "QVD2";
      =     M 1006.0;
NETWORK
TITLE =
      A     "QVD6";
      =     M 1006.1;
NETWORK
TITLE =
      A     "QVD3";
      =     M 1006.2;
NETWORK
TITLE =
      A     Q 6.3;
      =     M 1006.3;
NETWORK
TITLE =
      A     "QVD4";
      =     M 1006.4;
NETWORK
TITLE =
      A     Q 6.5;
      =     M 1006.5;
NETWORK
TITLE =
      A     "QVD5";
      =     M 1006.6;
NETWORK
TITLE =
      A     Q 6.7;
      =     M 1006.7;
NETWORK
TITLE =
      A     Q 7.0;
      =     M 1007.0;
NETWORK
TITLE =
      A     Q 7.1;
      =     M 1007.1;
NETWORK
TITLE =
      A     Q 7.2;
      =     M 1007.2;
NETWORK
TITLE =
      A     Q 7.3;
      =     M 1007.3;
NETWORK
TITLE =
      A     Q 7.4;
      =     M 1007.4;
NETWORK
TITLE =
      A     Q 7.5;
      =     M 1007.5;
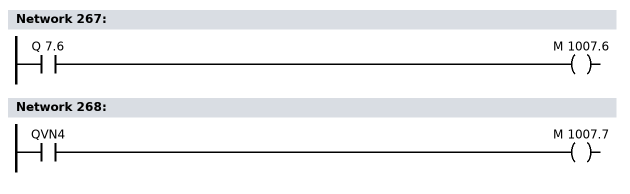
NETWORK
TITLE =
      A     Q 7.6;
      =     M 1007.6;
NETWORK
TITLE =
      A     "QVN4";
      =     M 1007.7;
END_FUNCTION_BLOCK

FUNCTION "DO_MANUAL" : VOID	// FC 1
VERSION : 0.1
VAR_INPUT
  MANUAL : BOOL ;
  PUSK : BOOL ;
  STOP : BOOL ;
END_VAR
VAR_OUTPUT
  M_DO : BOOL ;
END_VAR
BEGIN
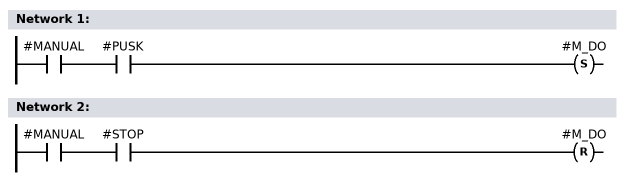
NETWORK
TITLE =
      A     #MANUAL;
      A     #PUSK;
      S     #M_DO;
NETWORK
TITLE =
      A     #MANUAL;
      A     #STOP;
      R     #M_DO;
END_FUNCTION

DATA_BLOCK DB 1
VERSION : 0.0
"DI_DO_STATE"
BEGIN
END_DATA_BLOCK

DATA_BLOCK DB 14
AUTHOR : SIMATIC
FAMILY : COM_FUNC
VERSION : 0.0
"GET"
BEGIN
END_DATA_BLOCK

DATA_BLOCK DB 15
AUTHOR : SIMATIC
FAMILY : COM_FUNC
VERSION : 0.0
"PUT"
BEGIN
END_DATA_BLOCK

ORGANIZATION_BLOCK OB 1
TITLE = "Main Program Sweep (Cycle)"
VERSION : 0.1
VAR_TEMP
  OB1_EV_CLASS : BYTE ;	//Bits 0-3 = 1 (Coming event), Bits 4-7 = 1 (Event class 1)
  OB1_SCAN_1 : BYTE ;	//1 (Cold restart scan 1 of OB 1), 3 (Scan 2-n of OB 1)
  OB1_PRIORITY : BYTE ;	//Priority of OB Execution
  OB1_OB_NUMBR : BYTE ;	//1 (Organization block 1, OB1)
  OB1_RESERVED_1 : BYTE ;	//Reserved for system
  OB1_RESERVED_2 : BYTE ;	//Reserved for system
  OB1_PREV_CYCLE : INT ;	//Cycle time of previous OB1 scan (milliseconds)
  OB1_MIN_CYCLE : INT ;	//Minimum cycle time of OB1 (milliseconds)
  OB1_MAX_CYCLE : INT ;	//Maximum cycle time of OB1 (milliseconds)
  OB1_DATE_TIME : DATE_AND_TIME ;	//Date and time OB1 started
  bypass : BOOL ;
  not_use : BOOL ;
  NV26_Hi_LVL : REAL ;
  NV26_Low_LVL : REAL ;
  NV26_LVL : REAL ;
  NV26_LVL_di : DINT ;
END_VAR
BEGIN
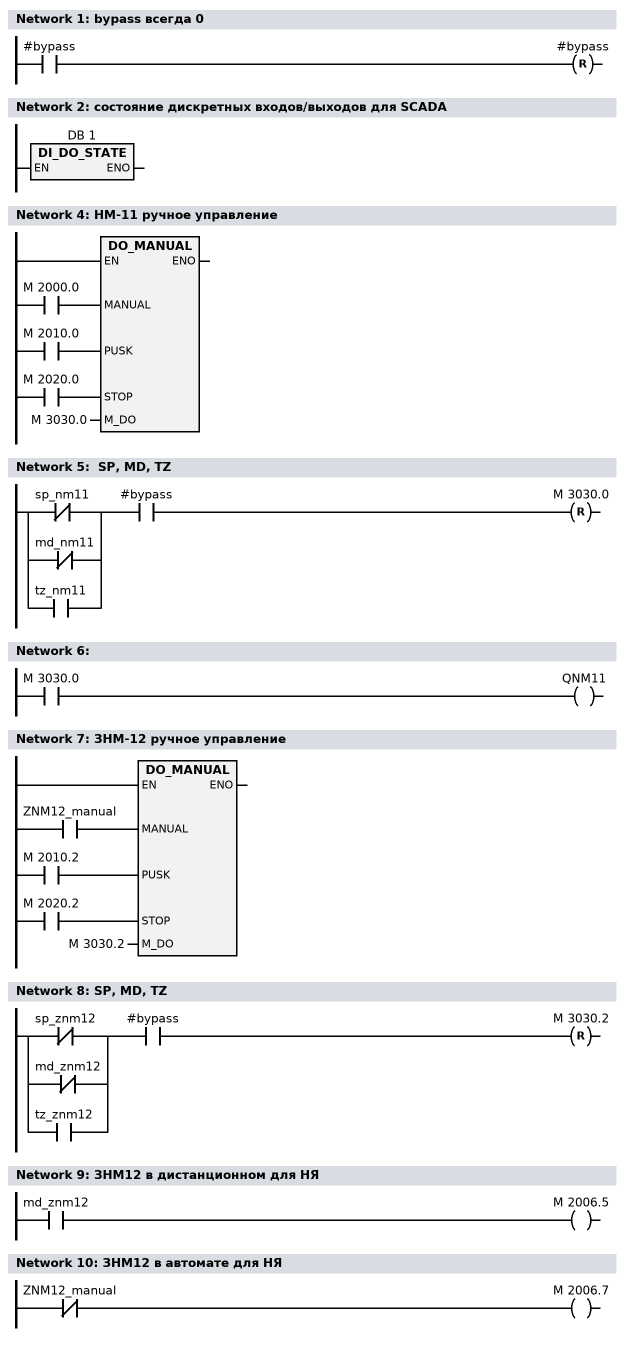
NETWORK
TITLE = bypass всегда 0
      A     #bypass;
      R     #bypass;
NETWORK
TITLE = состояние дискретных входов/выходов для SCADA
      CALL  "DI_DO_STATE" , DB 1;
      NOP   0;
NETWORK
TITLE = Прочитать по сети значения из ПЛК КИП
      A     M 100.3;
      =     L 38.0;
      BLD   103;
      BLD   9;
      =     L 43.0;
      CDB;
      OPN   DI 14;
      TAR2  LD 39;
      A     L 38.0;
      =     DIX 0.0;
      L     1;
      T     DIW 2;
      L     W#16#1002;
      T     DIW 8;
      L     120;
      T     DIW 10;
      L     0;
      T     DIW 12;
      L     P#M 1000.0;
      T     DID 14;
      L     W#16#1002;
      T     DIW 48;
      L     120;
      T     DIW 50;
      L     0;
      T     DIW 52;
      L     P#M 4000.0;
      T     DID 54;
      LAR2  P#DBX 0.0;
      UC    "GET";
      LAR2  LD 39;
      CDB;
      BLD   10;
      NOP   0;
NETWORK
TITLE = НМ-11 ручное управление
      A     M 2000.0;
      =     L 38.0;
      BLD   103;
      A     M 2010.0;
      =     L 38.1;
      BLD   103;
      A     M 2020.0;
      =     L 38.2;
      BLD   103;
      CALL  "DO_MANUAL" (
           MANUAL                   := L 38.0,
           PUSK                     := L 38.1,
           STOP                     := L 38.2,
           M_DO                     := M 3030.0);
      NOP   0;
NETWORK
TITLE =  SP, MD, TZ 
//Контроль живлення, місцеве/дистанційне, тепловий захист
      A(;
      ON    "sp_nm11";
      ON    "md_nm11";
      O     "tz_nm11";
      );
      A     #bypass;
      R     M 3030.0;
NETWORK
TITLE =
      A     M 3030.0;
      =     "QNM11";
NETWORK
TITLE = ЗНМ-12 ручное управление
      A     "ZNM12_manual";
      =     L 38.0;
      BLD   103;
      A     M 2010.2;
      =     L 38.1;
      BLD   103;
      A     M 2020.2;
      =     L 38.2;
      BLD   103;
      CALL  "DO_MANUAL" (
           MANUAL                   := L 38.0,
           PUSK                     := L 38.1,
           STOP                     := L 38.2,
           M_DO                     := M 3030.2);
      NOP   0;
NETWORK
TITLE = SP, MD, TZ
      A(;
      ON    "sp_znm12";
      ON    "md_znm12";
      O     "tz_znm12";
      );
      A     #bypass;
      R     M 3030.2;
NETWORK
TITLE = ЗНМ12 в дистанционном для НЯ
      A     "md_znm12";
      =     M 2006.5;
NETWORK
TITLE = ЗНМ12 в автомате для НЯ
      AN    "ZNM12_manual";
      =     M 2006.7;
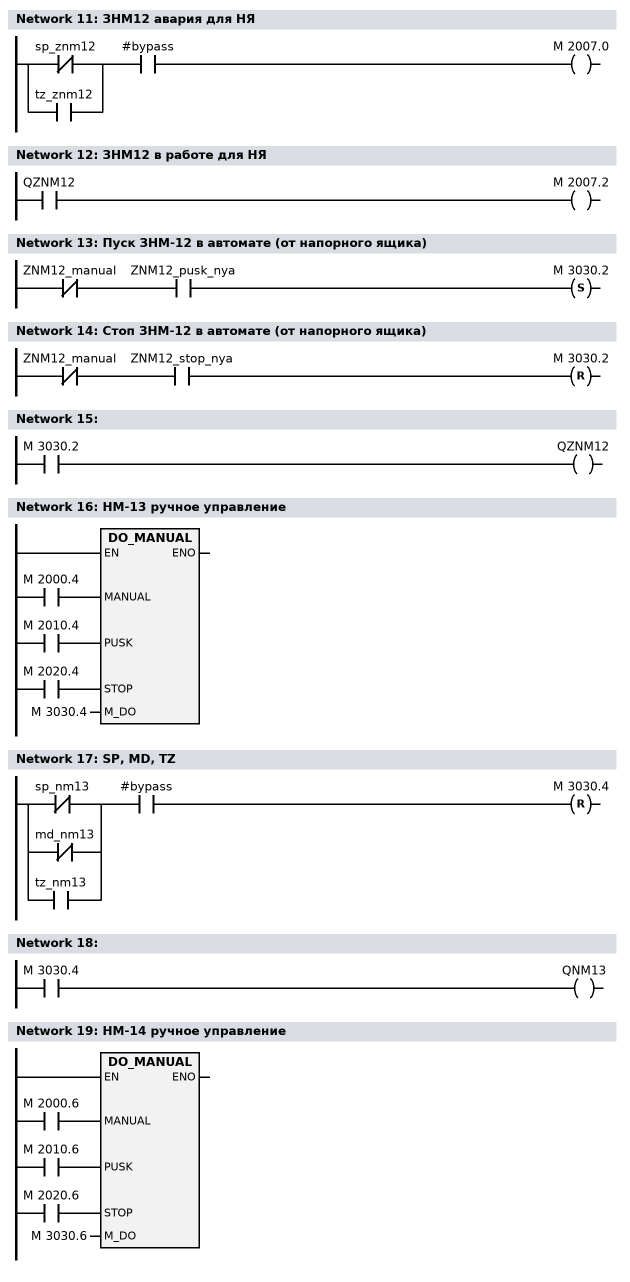
NETWORK
TITLE = ЗНМ12 авария для НЯ
      A(;
      ON    "sp_znm12";
      O     "tz_znm12";
      );
      A     #bypass;
      =     M 2007.0;
NETWORK
TITLE = ЗНМ12 в работе для НЯ
      A     "QZNM12";
      =     M 2007.2;
NETWORK
TITLE = Пуск ЗНМ-12 в автомате (от напорного ящика)
      AN    "ZNM12_manual";
      A     "ZNM12_pusk_nya";
      S     M 3030.2;
NETWORK
TITLE = Стоп ЗНМ-12 в автомате (от напорного ящика)
      AN    "ZNM12_manual";
      A     "ZNM12_stop_nya";
      R     M 3030.2;
NETWORK
TITLE =
      A     M 3030.2;
      =     "QZNM12";
NETWORK
TITLE = НМ-13 ручное управление
      A     M 2000.4;
      =     L 38.0;
      BLD   103;
      A     M 2010.4;
      =     L 38.1;
      BLD   103;
      A     M 2020.4;
      =     L 38.2;
      BLD   103;
      CALL  "DO_MANUAL" (
           MANUAL                   := L 38.0,
           PUSK                     := L 38.1,
           STOP                     := L 38.2,
           M_DO                     := M 3030.4);
      NOP   0;
NETWORK
TITLE = SP, MD, TZ
      A(;
      ON    "sp_nm13";
      ON    "md_nm13";
      O     "tz_nm13";
      );
      A     #bypass;
      R     M 3030.4;
NETWORK
TITLE =
      A     M 3030.4;
      =     "QNM13";
NETWORK
TITLE = НМ-14 ручное управление
      A     M 2000.6;
      =     L 38.0;
      BLD   103;
      A     M 2010.6;
      =     L 38.1;
      BLD   103;
      A     M 2020.6;
      =     L 38.2;
      BLD   103;
      CALL  "DO_MANUAL" (
           MANUAL                   := L 38.0,
           PUSK                     := L 38.1,
           STOP                     := L 38.2,
           M_DO                     := M 3030.6);
      NOP   0;
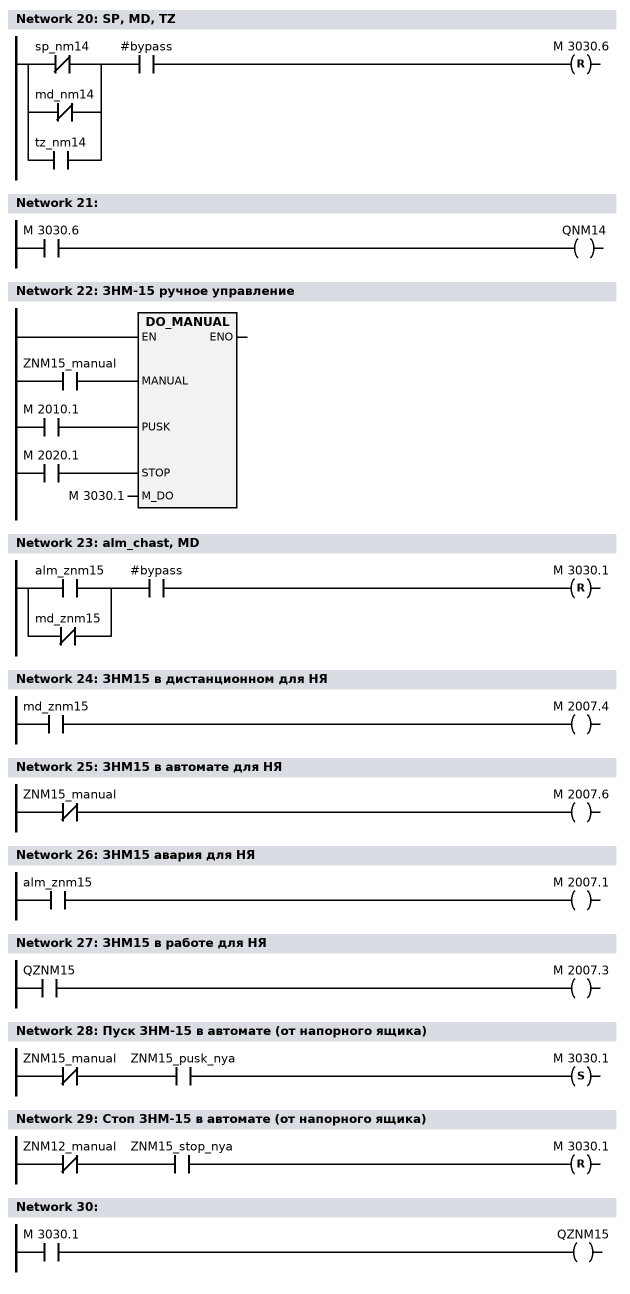
NETWORK
TITLE = SP, MD, TZ 
      A(;
      ON    "sp_nm14";
      ON    "md_nm14";
      O     "tz_nm14";
      );
      A     #bypass;
      R     M 3030.6;
NETWORK
TITLE =
      A     M 3030.6;
      =     "QNM14";
NETWORK
TITLE = ЗНМ-15 ручное управление
      A     "ZNM15_manual";
      =     L 38.0;
      BLD   103;
      A     M 2010.1;
      =     L 38.1;
      BLD   103;
      A     M 2020.1;
      =     L 38.2;
      BLD   103;
      CALL  "DO_MANUAL" (
           MANUAL                   := L 38.0,
           PUSK                     := L 38.1,
           STOP                     := L 38.2,
           M_DO                     := M 3030.1);
      NOP   0;
NETWORK
TITLE = alm_chast, MD
      A(;
      O     "alm_znm15";
      ON    "md_znm15";
      );
      A     #bypass;
      R     M 3030.1;
NETWORK
TITLE = ЗНМ15 в дистанционном для НЯ
      A     "md_znm15";
      =     M 2007.4;
NETWORK
TITLE = ЗНМ15 в автомате для НЯ
      AN    "ZNM15_manual";
      =     M 2007.6;
NETWORK
TITLE = ЗНМ15 авария для НЯ
      A     "alm_znm15";
      =     M 2007.1;
NETWORK
TITLE = ЗНМ15 в работе для НЯ
      A     "QZNM15";
      =     M 2007.3;
NETWORK
TITLE = Пуск ЗНМ-15 в автомате (от напорного ящика)
      AN    "ZNM15_manual";
      A     "ZNM15_pusk_nya";
      S     M 3030.1;
NETWORK
TITLE = Стоп ЗНМ-15 в автомате (от напорного ящика)
      AN    "ZNM12_manual";
      A     "ZNM15_stop_nya";
      R     M 3030.1;
NETWORK
TITLE =
      A     M 3030.1;
      =     "QZNM15";
